PROGRAM pouStation4
VAR
	stationMode: FB_Mode;
	tCalcNumberOfPages: REAL;
	ceil: REAL;
	PartBuild: FB_PartBuild;
	retvall: UDINT;
	// TODO
	tPartPresent: BOOL;
	stationPower: FB_PowerDelay;
END_VAR

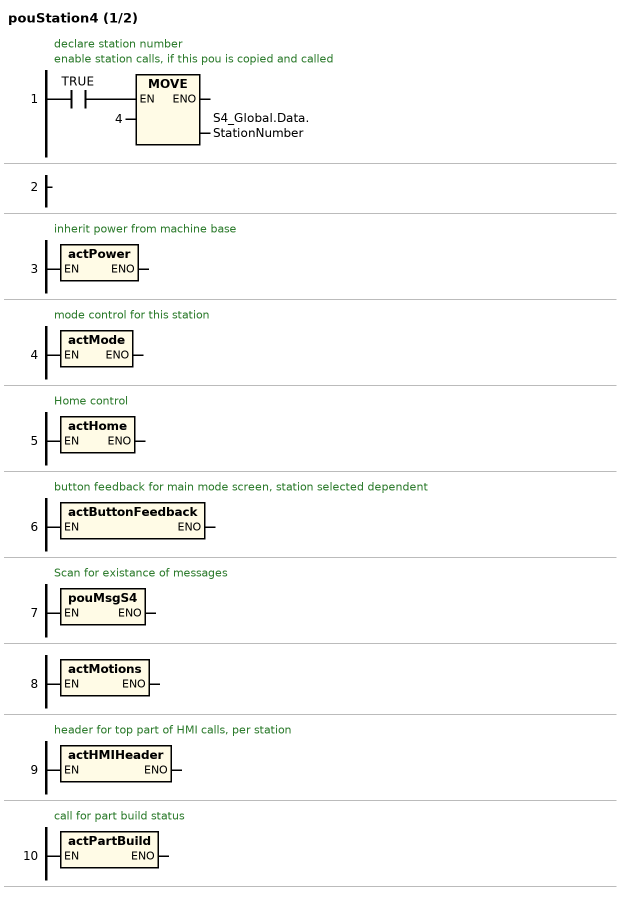
// NETWORK 1
// declare station number
// enable station calls, if this pou is copied and called
S4_Global.Data.StationNumber := 4;

// NETWORK 2

// NETWORK 3
// inherit power from machine base
actPower();

// NETWORK 4
// mode control for this station
actMode();

// NETWORK 5
// Home control
actHome();

// NETWORK 6
// button feedback for main mode screen, station selected dependent
actButtonFeedback();

// NETWORK 7
// Scan for existance of messages
pouMsgS4();

// NETWORK 8
actMotions();

// NETWORK 9
// header for top part of HMI calls, per station
actHMIHeader();

// NETWORK 10
// call for part build status
actPartBuild();

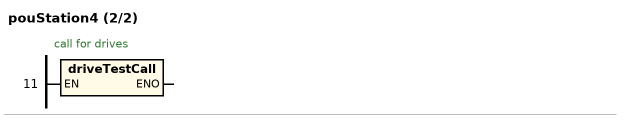
// NETWORK 11
// call for drives
driveTestCall();

ACTION actButtonFeedback:
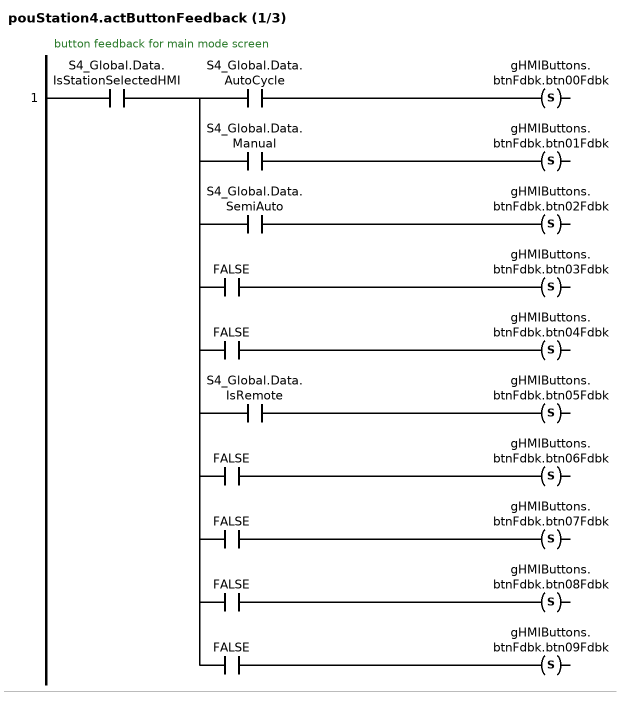
// NETWORK 1
// button feedback for main mode screen
gHMIButtons.btnFdbk.btn00Fdbk S= S4_Global.Data.IsStationSelectedHMI AND S4_Global.Data.AutoCycle;
gHMIButtons.btnFdbk.btn01Fdbk S= S4_Global.Data.IsStationSelectedHMI AND S4_Global.Data.Manual;
gHMIButtons.btnFdbk.btn02Fdbk S= S4_Global.Data.IsStationSelectedHMI AND S4_Global.Data.SemiAuto;
gHMIButtons.btnFdbk.btn03Fdbk S= S4_Global.Data.IsStationSelectedHMI AND FALSE;
gHMIButtons.btnFdbk.btn04Fdbk S= S4_Global.Data.IsStationSelectedHMI AND FALSE;
gHMIButtons.btnFdbk.btn05Fdbk S= S4_Global.Data.IsStationSelectedHMI AND S4_Global.Data.IsRemote;
gHMIButtons.btnFdbk.btn06Fdbk S= S4_Global.Data.IsStationSelectedHMI AND FALSE;
gHMIButtons.btnFdbk.btn07Fdbk S= S4_Global.Data.IsStationSelectedHMI AND FALSE;
gHMIButtons.btnFdbk.btn08Fdbk S= S4_Global.Data.IsStationSelectedHMI AND FALSE;
gHMIButtons.btnFdbk.btn09Fdbk S= S4_Global.Data.IsStationSelectedHMI AND FALSE;

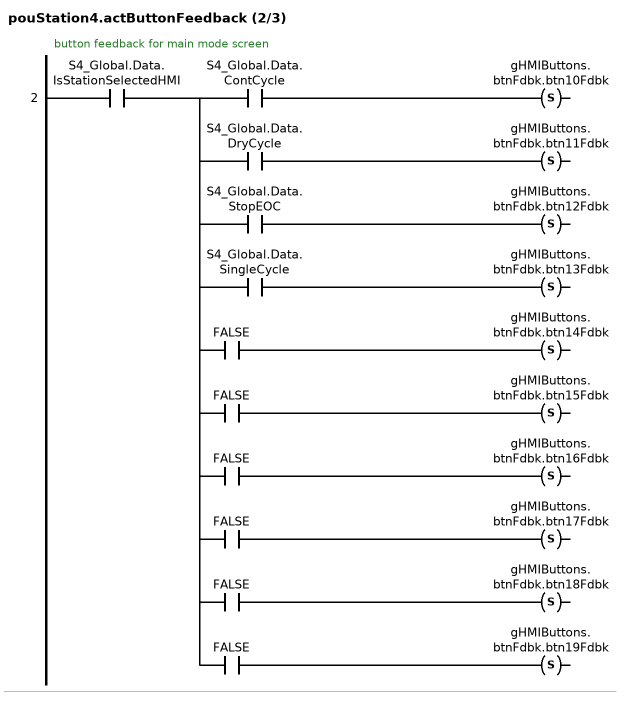
// NETWORK 2
// button feedback for main mode screen
gHMIButtons.btnFdbk.btn10Fdbk S= S4_Global.Data.IsStationSelectedHMI AND S4_Global.Data.ContCycle;
gHMIButtons.btnFdbk.btn11Fdbk S= S4_Global.Data.IsStationSelectedHMI AND S4_Global.Data.DryCycle;
gHMIButtons.btnFdbk.btn12Fdbk S= S4_Global.Data.IsStationSelectedHMI AND S4_Global.Data.StopEOC;
gHMIButtons.btnFdbk.btn13Fdbk S= S4_Global.Data.IsStationSelectedHMI AND S4_Global.Data.SingleCycle;
gHMIButtons.btnFdbk.btn14Fdbk S= S4_Global.Data.IsStationSelectedHMI AND FALSE;
gHMIButtons.btnFdbk.btn15Fdbk S= S4_Global.Data.IsStationSelectedHMI AND FALSE;
gHMIButtons.btnFdbk.btn16Fdbk S= S4_Global.Data.IsStationSelectedHMI AND FALSE;
gHMIButtons.btnFdbk.btn17Fdbk S= S4_Global.Data.IsStationSelectedHMI AND FALSE;
gHMIButtons.btnFdbk.btn18Fdbk S= S4_Global.Data.IsStationSelectedHMI AND FALSE;
gHMIButtons.btnFdbk.btn19Fdbk S= S4_Global.Data.IsStationSelectedHMI AND FALSE;

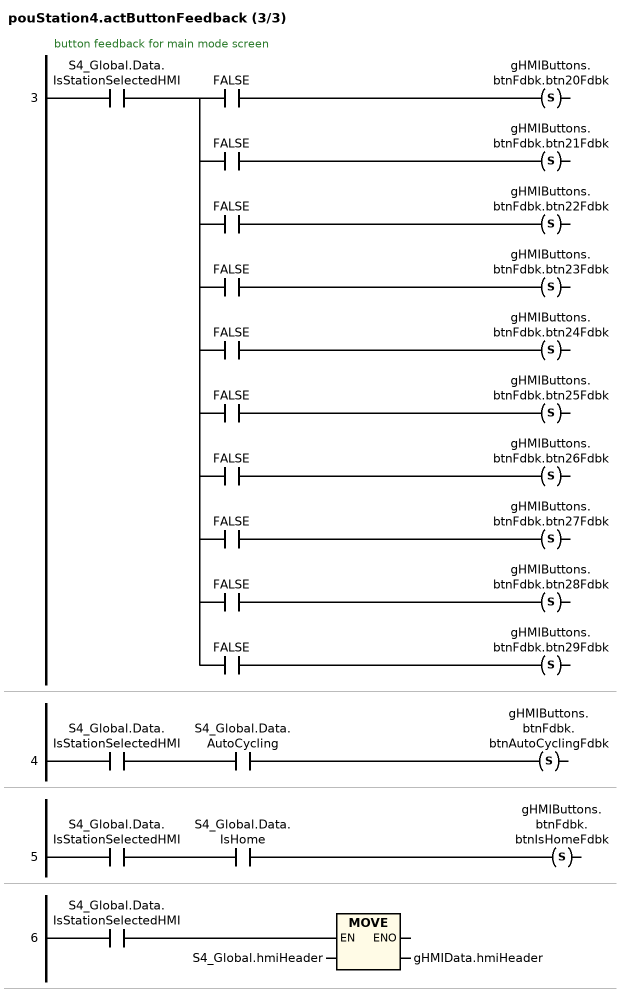
// NETWORK 3
// button feedback for main mode screen
gHMIButtons.btnFdbk.btn20Fdbk S= S4_Global.Data.IsStationSelectedHMI AND FALSE;
gHMIButtons.btnFdbk.btn21Fdbk S= S4_Global.Data.IsStationSelectedHMI AND FALSE;
gHMIButtons.btnFdbk.btn22Fdbk S= S4_Global.Data.IsStationSelectedHMI AND FALSE;
gHMIButtons.btnFdbk.btn23Fdbk S= S4_Global.Data.IsStationSelectedHMI AND FALSE;
gHMIButtons.btnFdbk.btn24Fdbk S= S4_Global.Data.IsStationSelectedHMI AND FALSE;
gHMIButtons.btnFdbk.btn25Fdbk S= S4_Global.Data.IsStationSelectedHMI AND FALSE;
gHMIButtons.btnFdbk.btn26Fdbk S= S4_Global.Data.IsStationSelectedHMI AND FALSE;
gHMIButtons.btnFdbk.btn27Fdbk S= S4_Global.Data.IsStationSelectedHMI AND FALSE;
gHMIButtons.btnFdbk.btn28Fdbk S= S4_Global.Data.IsStationSelectedHMI AND FALSE;
gHMIButtons.btnFdbk.btn29Fdbk S= S4_Global.Data.IsStationSelectedHMI AND FALSE;

// NETWORK 4
gHMIButtons.btnFdbk.btnAutoCyclingFdbk S= S4_Global.Data.IsStationSelectedHMI AND S4_Global.Data.AutoCycling;

// NETWORK 5
gHMIButtons.btnFdbk.btnIsHomeFdbk S= S4_Global.Data.IsStationSelectedHMI AND S4_Global.Data.IsHome;

// NETWORK 6
IF S4_Global.Data.IsStationSelectedHMI THEN gHMIData.hmiHeader := S4_Global.hmiHeader; END_IF
END_ACTION

ACTION actHMIHeader:
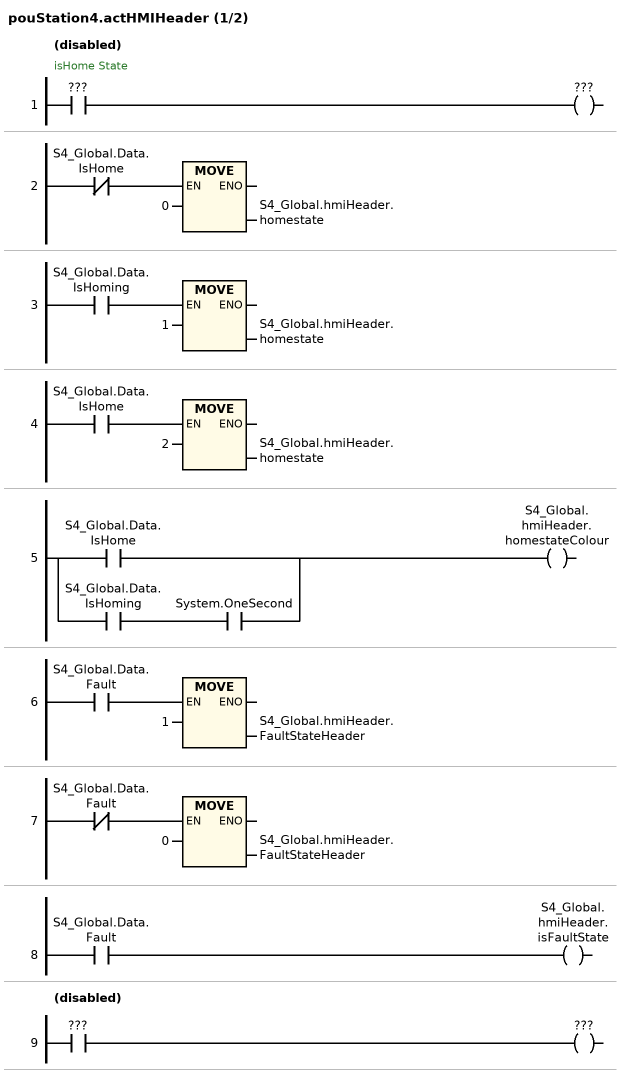
// NETWORK 1 (disabled)
// isHome State
// ??? := ???;

// NETWORK 2
IF NOT S4_Global.Data.IsHome THEN S4_Global.hmiHeader.homestate := 0; END_IF

// NETWORK 3
IF S4_Global.Data.IsHoming THEN S4_Global.hmiHeader.homestate := 1; END_IF

// NETWORK 4
IF S4_Global.Data.IsHome THEN S4_Global.hmiHeader.homestate := 2; END_IF

// NETWORK 5
S4_Global.hmiHeader.homestateColour := S4_Global.Data.IsHome OR S4_Global.Data.IsHoming AND System.OneSecond;

// NETWORK 6
IF S4_Global.Data.Fault THEN S4_Global.hmiHeader.FaultStateHeader := 1; END_IF

// NETWORK 7
IF NOT S4_Global.Data.Fault THEN S4_Global.hmiHeader.FaultStateHeader := 0; END_IF

// NETWORK 8
S4_Global.hmiHeader.isFaultState := S4_Global.Data.Fault;

// NETWORK 9 (disabled)
// ??? := ???;

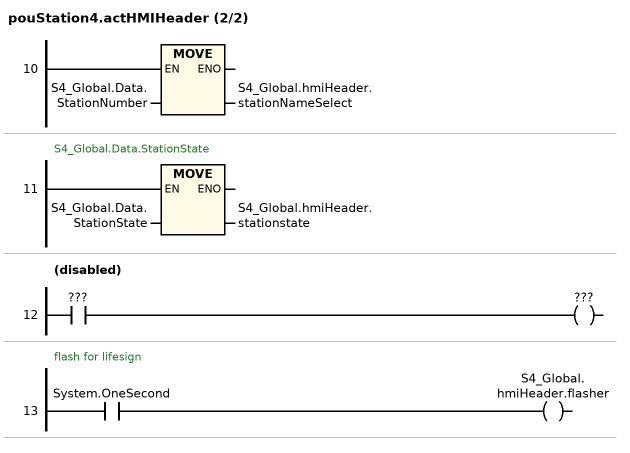
// NETWORK 10
S4_Global.hmiHeader.stationNameSelect := S4_Global.Data.StationNumber;

// NETWORK 11
// S4_Global.Data.StationState
S4_Global.hmiHeader.stationstate := S4_Global.Data.StationState;

// NETWORK 12 (disabled)
// ??? := ???;

// NETWORK 13
// flash for lifesign
S4_Global.hmiHeader.flasher := System.OneSecond;
END_ACTION

ACTION actHome:
//Set home status for station

IF 
//are all motions returned
S4_01_Motion_01_01.Motion.qReturnDepth AND
S4_01_Motion_01_02.Motion.qReturnDepth AND
S4_01_Motion_01_03.Motion.qReturnDepth AND
S4_01_Motion_01_04.Motion.qReturnDepth AND
S4_01_Motion_01_05.Motion.qReturnDepth AND
S4_01_Motion_01_06.Motion.qReturnDepth

	THEN
		//set IsHome value for station
		S4_Global.Data.IsHome := TRUE;
	ELSE
		S4_Global.Data.IsHome := FALSE;
END_IF
END_ACTION

ACTION actMaxNumStationPages:
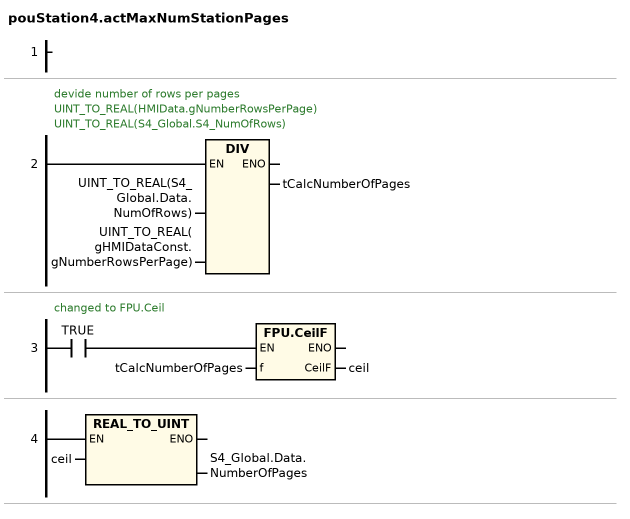
// NETWORK 1

// NETWORK 2
// devide number of rows per pages
// UINT_TO_REAL(HMIData.gNumberRowsPerPage)
// UINT_TO_REAL(S4_Global.S4_NumOfRows)
tCalcNumberOfPages := (UINT_TO_REAL(S4_Global.Data.NumOfRows)) / (UINT_TO_REAL(gHMIDataConst.gNumberRowsPerPage));

// NETWORK 3
// changed to FPU.Ceil
ceil := FPU.CeilF(f := tCalcNumberOfPages);

// NETWORK 4
S4_Global.Data.NumberOfPages := REAL_TO_UINT(ceil);
END_ACTION

ACTION actMode:
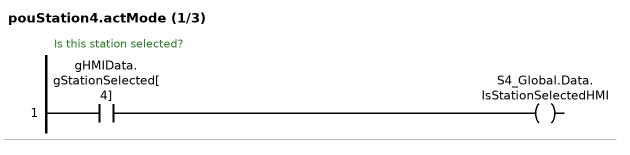
// NETWORK 1
// Is this station selected?
S4_Global.Data.IsStationSelectedHMI := gHMIData.gStationSelected[4];

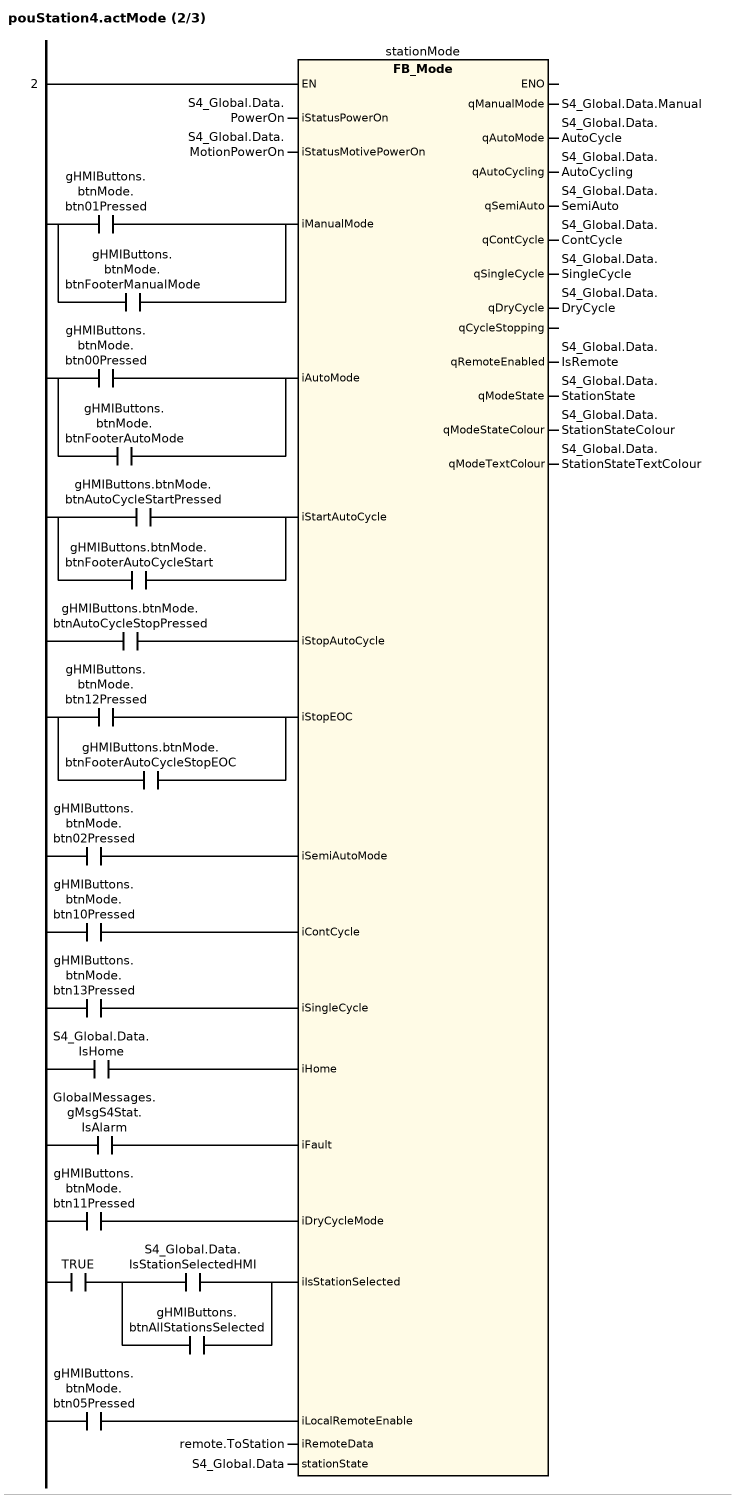
// NETWORK 2
stationMode(
    iStatusPowerOn := S4_Global.Data.PowerOn,
    iStatusMotivePowerOn := S4_Global.Data.MotionPowerOn,
    iManualMode := gHMIButtons.btnMode.btn01Pressed OR gHMIButtons.btnMode.btnFooterManualMode,
    iAutoMode := gHMIButtons.btnMode.btn00Pressed OR gHMIButtons.btnMode.btnFooterAutoMode,
    iStartAutoCycle := gHMIButtons.btnMode.btnAutoCycleStartPressed OR gHMIButtons.btnMode.btnFooterAutoCycleStart,
    iStopAutoCycle := gHMIButtons.btnMode.btnAutoCycleStopPressed,
    iStopEOC := gHMIButtons.btnMode.btn12Pressed OR gHMIButtons.btnMode.btnFooterAutoCycleStopEOC,
    iSemiAutoMode := gHMIButtons.btnMode.btn02Pressed,
    iContCycle := gHMIButtons.btnMode.btn10Pressed,
    iSingleCycle := gHMIButtons.btnMode.btn13Pressed,
    iHome := S4_Global.Data.IsHome,
    iFault := GlobalMessages.gMsgS4Stat.IsAlarm,
    iDryCycleMode := gHMIButtons.btnMode.btn11Pressed,
    iIsStationSelected := TRUE AND (S4_Global.Data.IsStationSelectedHMI OR gHMIButtons.btnAllStationsSelected),
    iLocalRemoteEnable := gHMIButtons.btnMode.btn05Pressed,
    iRemoteData := remote.ToStation,
    stationState := S4_Global.Data,
    qManualMode => S4_Global.Data.Manual,
    qAutoMode => S4_Global.Data.AutoCycle,
    qAutoCycling => S4_Global.Data.AutoCycling,
    qSemiAuto => S4_Global.Data.SemiAuto,
    qContCycle => S4_Global.Data.ContCycle,
    qSingleCycle => S4_Global.Data.SingleCycle,
    qDryCycle => S4_Global.Data.DryCycle,
    qRemoteEnabled => S4_Global.Data.IsRemote,
    qModeState => S4_Global.Data.StationState,
    qModeStateColour => S4_Global.Data.StationStateColour,
    qModeTextColour => S4_Global.Data.StationStateTextColour); // FB_Mode

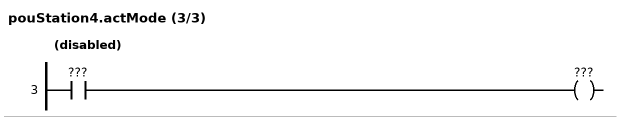
// NETWORK 3 (disabled)
// ??? := ???;
END_ACTION

ACTION actMotions:
//station 1 = 10000 index


//init number of rows
S4_Global.Data.NumOfRows := 0;

//page 1
S4_01_Motion_01_01();
S4_01_Motion_01_02();
S4_01_Motion_01_03();
S4_01_Motion_01_04();
S4_01_Motion_01_05();
S4_01_Motion_01_06();

//page 2
S4_01_Motion_02_07();
S4_01_Motion_02_08();
S4_01_Motion_02_09();
S4_01_Motion_02_10();
S4_01_Motion_02_11();
S4_01_Motion_02_12();

//page 3
S4_01_Motion_03_13();
S4_01_Motion_03_14();
S4_01_Motion_03_15();
S4_01_Motion_03_16();
S4_01_Motion_03_17();
S4_01_Motion_03_18();

//page 4
S4_01_Motion_04_19();
S4_01_Motion_04_20();
S4_01_Motion_04_21();
S4_01_Motion_04_22();
S4_01_Motion_04_23();
S4_01_Motion_04_24();

//page 5
S4_01_Motion_05_25();
S4_01_Motion_05_26();
S4_01_Motion_05_27();
S4_01_Motion_05_28();
S4_01_Motion_05_29();
S4_01_Motion_05_30();

//page 6
S4_01_Motion_06_31();
S4_01_Motion_06_32();
S4_01_Motion_06_33();
S4_01_Motion_06_34();
S4_01_Motion_06_35();
S4_01_Motion_06_36();

//must be called after motionRow calls
actMaxNumStationPages();
END_ACTION

ACTION actPartBuild:
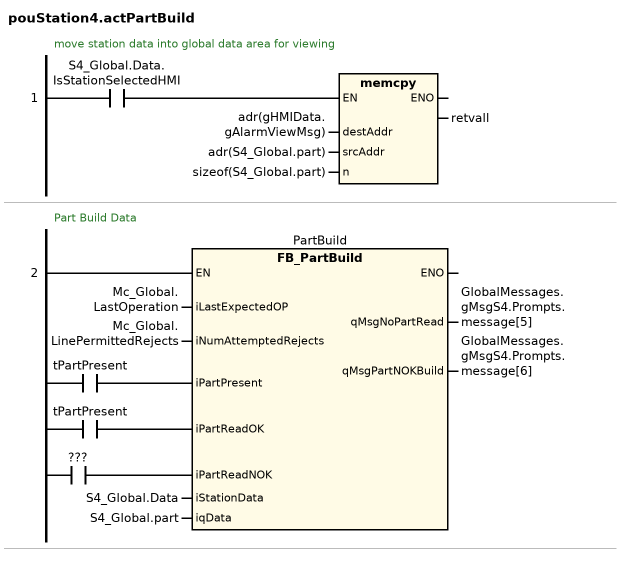
// NETWORK 1
// move station data into global data area for viewing
IF S4_Global.Data.IsStationSelectedHMI THEN
    retvall := memcpy(destAddr := adr(gHMIData.gAlarmViewMsg), srcAddr := adr(S4_Global.part), n := sizeof(S4_Global.part));
END_IF

// NETWORK 2
// Part Build Data
PartBuild(
    iLastExpectedOP := Mc_Global.LastOperation,
    iNumAttemptedRejects := Mc_Global.LinePermittedRejects,
    iPartPresent := tPartPresent,
    iPartReadOK := tPartPresent,
    iStationData := S4_Global.Data,
    iqData := S4_Global.part,
    qMsgNoPartRead => GlobalMessages.gMsgS4.Prompts.message[5],
    qMsgPartNOKBuild => GlobalMessages.gMsgS4.Prompts.message[6]); // FB_PartBuild
END_ACTION

ACTION actPower:
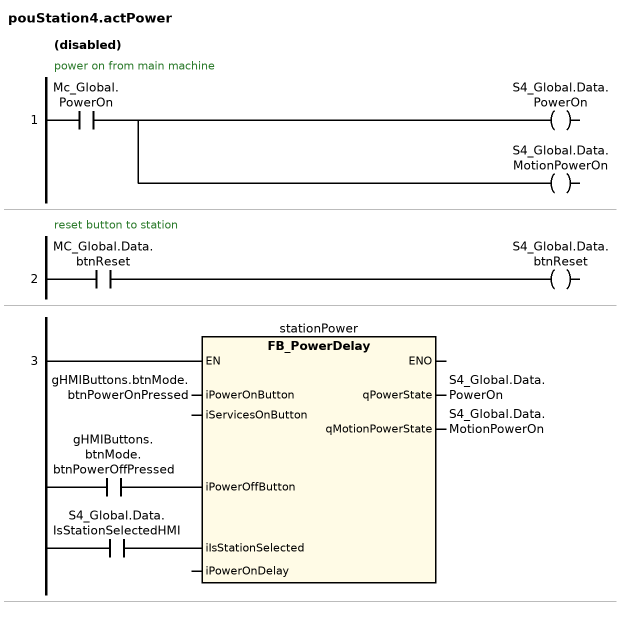
// NETWORK 1 (disabled)
// power on from main machine
// S4_Global.Data.PowerOn := Mc_Global.PowerOn;
// S4_Global.Data.MotionPowerOn := Mc_Global.PowerOn;

// NETWORK 2
// reset button to station
S4_Global.Data.btnReset := MC_Global.Data.btnReset;

// NETWORK 3
stationPower(
    iPowerOnButton := gHMIButtons.btnMode.btnPowerOnPressed,
    iPowerOffButton := gHMIButtons.btnMode.btnPowerOffPressed,
    iIsStationSelected := S4_Global.Data.IsStationSelectedHMI,
    qPowerState => S4_Global.Data.PowerOn,
    qMotionPowerState => S4_Global.Data.MotionPowerOn); // FB_PowerDelay
END_ACTION

END_PROGRAM

(* stored: Version 1.1.0.1, ProductVersion 3.1.4024.12
   POU pouStation4: Id {0041c954-93b0-4883-a4fc-8abf361a50dc}, SpecialFunc None
   Action actButtonFeedback: Id {008c04e6-8f55-4817-becc-ea8b21c78cfe}
   Action actHMIHeader: Id {b1f356cf-dab0-43e5-bc7e-04cd9aee677d}
   Action actHome: Id {819117c8-b6e8-4710-a5f5-acfc34bb4626}
   Action actMaxNumStationPages: Id {4e626d6a-996a-4dd3-aa5a-2c2903d5613e}
   Action actMode: Id {c36563c9-f500-4619-98b5-dc625fb8edfc}
   Action actMotions: Id {6bf7037e-d7f6-4ece-8f6b-94501b187b80}
   Action actPartBuild: Id {ab9ba25d-5531-4db0-8f7a-d75c06c7b310}
   Action actPower: Id {2903002e-2e03-4c68-bbbb-053a23d921cb} *)
